Staubli VAL3: Control_Joint.pgx

public program Control_Joint(jointRx& x_jJ)
  local string l_sItem[6]
  local num l_nNum
  local num l_nKey
  local num l_nData[6]
  local num l_nSelectIndex
begin

  //修改点位的 joint



  l_nData[0]=x_jJ.j1
  l_nData[1]=x_jJ.j2
  l_nData[2]=x_jJ.j3
  l_nData[3]=x_jJ.j4
  l_nData[4]=x_jJ.j5
  l_nData[5]=x_jJ.j6

  for l_nNum=0 to 5
    l_sItem[l_nNum]="j"+toString("",l_nNum+1)+"   :"+toString(".3",l_nData[l_nNum])
  endFor

  call Control_BottomS(",,,,,,取消,确定")
  call Control_PanelXY(8,0,15,6)
  call Control_Panel("Joint值")
  call Control_List(l_sItem,l_nSelectIndex)
  while true
    l_nKey=getKey()

    switch l_nKey
      case 261
        l_nSelectIndex=max(0,l_nSelectIndex-1)
      break

      case 266
        l_nSelectIndex=min(l_nSelectIndex+1,5)
      break

      case 278
        x_jJ.j1=l_nData[0]
        x_jJ.j2=l_nData[1]
        x_jJ.j3=l_nData[2]
        x_jJ.j4=l_nData[3]
        x_jJ.j5=l_nData[4]
        x_jJ.j6=l_nData[5]
        return
      break


      case 277,255
        return
      break

      case 270
        call Float_Edit(l_nData[l_nSelectIndex],nPanelLTopX+7,l_nSelectIndex+nPanelLTopY+1)
      break

    endSwitch

    if l_nKey!=-1
      for l_nNum=0 to 5
        l_sItem[l_nNum]="j"+toString("",l_nNum+1)+"   :"+toString(".3",l_nData[l_nNum])
      endFor
      call Control_List(l_sItem,l_nSelectIndex)

    endIf






  endWhile





end
